(* Logix 5000 project; controller KTC_PV_LAB1 vendor 1 type 14 code 150 rev 30.11; software revision 30.00 *)

TASK MainTask (continuous, watchdog 500 ms) : MainProgram

MODULES
   Local : vendor 1 type 14 code 150 (Compact 0, rev 30.11)
      Counters : Embedded (Compact 3, rev 1.1, Output RPI 20 ms)
      Discrete_IO : Embedded (Compact 1, rev 3.1, Output RPI 20 ms)
      Analog_IO : Embedded (Compact 2, rev 1.1, Output RPI 80 ms)
END_MODULES

PROGRAM MainProgram   (* main routine MainRoutine *)
VAR
   LED2 : ALIAS FOR Local:1:O.Data.1;   // RUN LIGHT 2
   LED_1 : ALIAS FOR Local:1:O.Data.0;   // RUN LIGHT
   LED_3 : ALIAS FOR Local:1:O.Data.3;   // PV RUN
   PB4 : ALIAS FOR Local:1:I.Data.9;   // STOP 2
   PB_1 : ALIAS FOR Local:1:I.Data.0;   // START
   PB_2 : ALIAS FOR Local:1:I.Data.8;   // STOP
   PB_3 : ALIAS FOR Local:1:I.Data.1;   // START 2
   PL_1 : ALIAS FOR Local:1:O.Data.0;   // ON LED
   PV_START : BOOL;
   PV_STOP : BOOL;
   SW_1 : BOOL;   // PV START
END_VAR

ROUTINE MainRoutine   (* ladder *)
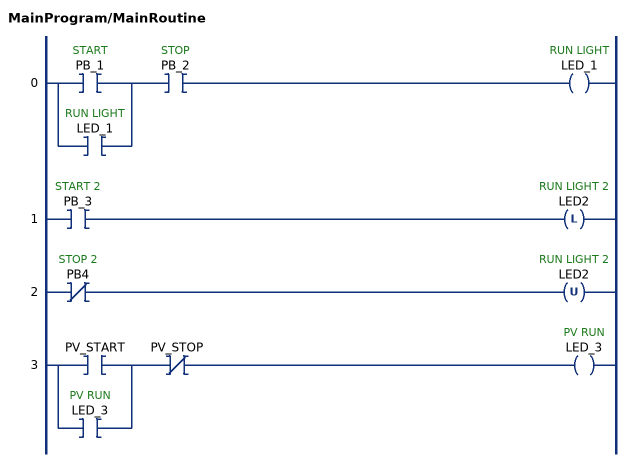
   0: [XIC(PB_1) ,XIC(LED_1) ]XIC(PB_2)OTE(LED_1);
   1: XIC(PB_3)OTL(LED2);
   2: XIO(PB4)OTU(LED2);
   3: [XIC(PV_START) ,XIC(LED_3) ]XIO(PV_STOP)OTE(LED_3);
END_ROUTINE
END_PROGRAM
